TYPE AxesMoveOutOfLimitSwitchProcessArgs :
STRUCT
	///Positive or negative limit switch
	switch: LimitSwitches;
END_STRUCT
END_TYPE

(* stored: Version 1.1.0.1, ProductVersion 3.1.4019.2
   DUT AxesMoveOutOfLimitSwitchProcessArgs: Id {2322d16d-911a-404c-a94b-cda3a9330b40} *)
